// TIA Portal project "Clase4" (V14)
// Equivalente del tutorial 1 del TIA Portal de Youtube

(* hardware
DEVICE "S7-1200 station_1"  S7-1200 Station
   slot 0: "Rack_0"  S7-1200 Rack  Rack  V1.0
   slot 1: "Limon_PLC"  CPU 1214C DC/DC/DC  6ES7 214-1AG40-0XB0  V4.2
DEVICE "S71500/ET200MP station_1"  S7-1500 station
   slot 0: "Rail_0"  Rack  6ES7 590-1***0-0AA0
   slot 1: "Limon 1516"  CPU 1516F-3 PN/DP  6ES7 516-3FN01-0AB0  V2.1
      slot 3: "CPU display_1"  6ES7591-1BA00-0AA0
   slot 2: "DI 32x24VDC HF_1"  DI 32x24VDC HF  6ES7 521-1BL00-0AB0  V2.1
   slot 3: "DQ 32x24VDC/0.5A HF_1"  DQ 32x24VDC/0.5A HF  6ES7 522-1BL01-0AB0  V1.0
   slot 4: "AI 8xU/I/RTD/TC ST_1"  AI 8xU/I/RTD/TC ST  6ES7 531-7KF00-0AB0  V2.1
   slot 5: "AQ 8xU/I HS_1"  AQ 8xU/I HS  6ES7 532-5HF00-0AB0  V2.1
*)

// ===== PLC "Limon_PLC"  CPU 1214C DC/DC/DC =====

VAR_GLOBAL   // PLC tag table "Default tag table"
   "start" AT %I0.0 : Bool;
   "stop" AT %I0.1 : Bool;
   "L1" AT %Q0.0 : Bool;
   "L2" AT %Q0.1 : Bool;
   "variable" AT %M2.0 : Bool;
   "sensor" AT %IW64 : Int;
   "variable_paso" AT %MD4 : Real;
   "lectura" AT %MW8 : Int;
END_VAR

FUNCTION "Arranque_Paro" : Void   // FC1, LAD
TITLE = Arranque y Paro
{ S7_Optimized_Access := 'TRUE' }
VERSION : 0.1
// Demostración de encendido y apagado de una lámpara con enclavamiento.
BEGIN

REGION Network 1: L1
   // Lámpara 1
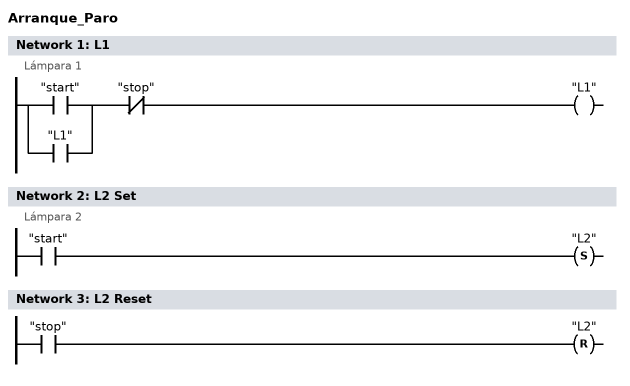
   RUNG wire#powerrail
      Contact( "start" )
      wire#w1
      I_Contact( "stop" )
      Coil( "L1" )
   END_RUNG
   RUNG wire#powerrail
      Contact( "L1" )
   END_RUNG wire#w1
   // the same network as SCL:
   "L1" := ("start" OR "L1") AND NOT "stop";
END_REGION

REGION Network 2: L2 Set
   // Lámpara 2
   RUNG wire#powerrail
      Contact( "start" )
      S_Coil( "L2" )
   END_RUNG
   // the same network as SCL:
   IF "start" THEN "L2" := TRUE; END_IF;
END_REGION

REGION Network 3: L2 Reset
   RUNG wire#powerrail
      Contact( "stop" )
      R_Coil( "L2" )
   END_RUNG
   // the same network as SCL:
   IF "stop" THEN "L2" := FALSE; END_IF;
END_REGION
END_FUNCTION

FUNCTION "Lectura Analogica" : Void   // FC2, LAD
{ S7_Optimized_Access := 'TRUE' }
VERSION : 0.1
BEGIN

REGION Network 1
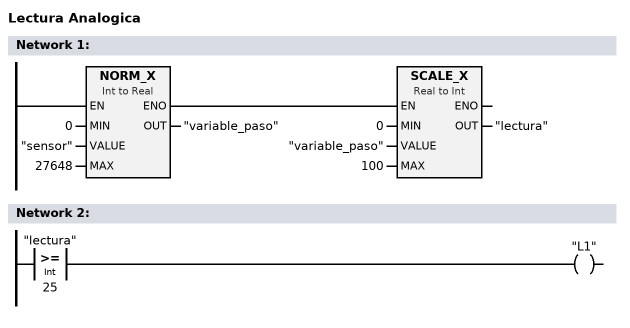
   RUNG wire#powerrail
      { S7_Templates := "[SrcType := Int, DestType := Real]" } Normalize(min := 0, value := "sensor", max := 27648, out => "variable_paso")
      { S7_Templates := "[SrcType := Real, DestType := Int]" } Scale(min := 0, value := "variable_paso", max := 100, out => "lectura")
   END_RUNG
   // the same network as SCL:
   "variable_paso" := NORM_X(MIN := 0, VALUE := "sensor", MAX := 27648);
   "lectura" := SCALE_X(MIN := 0, VALUE := "variable_paso", MAX := 100);
END_REGION

REGION Network 2
   RUNG wire#powerrail
      { S7_Templates := "SrcType := Int" } GE_Contact(in1 := "lectura", in2 := 25)
      Coil( "L1" )
   END_RUNG
   // the same network as SCL:
   "L1" := "lectura" >= 25;
END_REGION
END_FUNCTION

ORGANIZATION_BLOCK "Main"   // OB1, LAD, ProgramCycle
TITLE = "Main Program Sweep (Cycle)"
{ S7_Optimized_Access := 'TRUE' }
VERSION : 0.1
   VAR_INPUT
      Initial_Call : Bool;   // Initial call of this OB
      Remanence : Bool;   // =True, if remanent data are available
   END_VAR
BEGIN

REGION Network 1
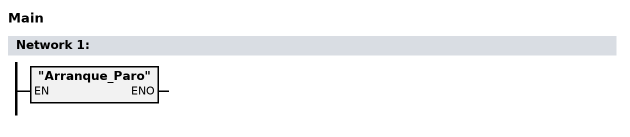
   RUNG wire#powerrail
      "Arranque_Paro"()
   END_RUNG
   // the same network as SCL:
   "Arranque_Paro"();
END_REGION
END_ORGANIZATION_BLOCK

// ===== PLC "Limon 1516"  CPU 1516F-3 PN/DP =====

VAR_GLOBAL   // PLC tag table "Default tag table"
   "inicio" AT %I0.0 : Bool;
   "paro" AT %I0.1 : Bool;
   "L1" AT %Q0.0 : Bool;
   "L2" AT %Q0.1 : Bool;
   "variable" AT %M2.0 : Bool;
   "System_Byte" AT %MB1 : Byte;
   "FirstScan" AT %M1.0 : Bool;
   "DiagStatusUpdate" AT %M1.1 : Bool;
   "AlwaysTRUE" AT %M1.2 : Bool;
   "AlwaysFALSE" AT %M1.3 : Bool;
   "Clock_Byte" AT %MB0 : Byte;
   "Clock_10Hz" AT %M0.0 : Bool;
   "Clock_5Hz" AT %M0.1 : Bool;
   "Clock_2.5Hz" AT %M0.2 : Bool;
   "Clock_2Hz" AT %M0.3 : Bool;
   "Clock_1.25Hz" AT %M0.4 : Bool;
   "Clock_1Hz" AT %M0.5 : Bool;
   "Clock_0.625Hz" AT %M0.6 : Bool;
   "Clock_0.5Hz" AT %M0.7 : Bool;
   "sensor" AT %IW12 : Int;
   "variable de paso" AT %MD18 : Real;
   "lectura" AT %MW22 : Int;
END_VAR

// folder: System blocks/Program resources

DATA_BLOCK "Timer1"   // DB1
{ S7_Optimized_Access := 'TRUE' }
AUTHOR : Simatic
FAMILY : IEC
NAME : IEC_TMR
VERSION : 1.0
// stored: InstanceOfName IEC_TIMER
"IEC_TIMER"
BEGIN
END_DATA_BLOCK

DATA_BLOCK "Timer2"   // DB2
{ S7_Optimized_Access := 'TRUE' }
AUTHOR : Simatic
FAMILY : IEC
NAME : IEC_TMR
VERSION : 1.0
// stored: InstanceOfName IEC_TIMER
"IEC_TIMER"
BEGIN
END_DATA_BLOCK

// folder: (top level)

FUNCTION "Arranque_Paro" : Void   // FC1, LAD
TITLE = Arranque y Paro
{ S7_Optimized_Access := 'TRUE' }
VERSION : 0.1
// Demostración de encendido y apagado de una lámpara con enclavamiento.
BEGIN

REGION Network 1: L1
   // Lámpara 1
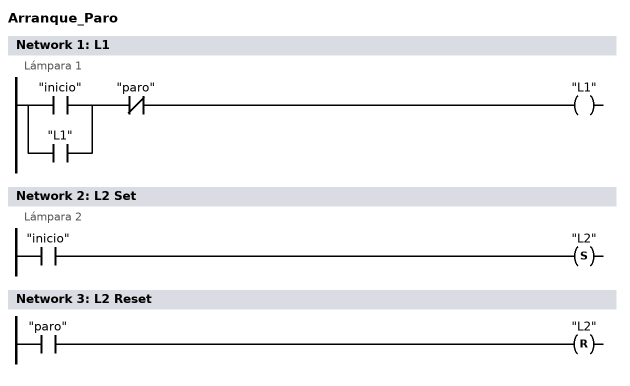
   RUNG wire#powerrail
      Contact( "inicio" )
      wire#w1
      I_Contact( "paro" )
      Coil( "L1" )
   END_RUNG
   RUNG wire#powerrail
      Contact( "L1" )
   END_RUNG wire#w1
   // the same network as SCL:
   "L1" := ("inicio" OR "L1") AND NOT "paro";
END_REGION

REGION Network 2: L2 Set
   // Lámpara 2
   RUNG wire#powerrail
      Contact( "inicio" )
      S_Coil( "L2" )
   END_RUNG
   // the same network as SCL:
   IF "inicio" THEN "L2" := TRUE; END_IF;
END_REGION

REGION Network 3: L2 Reset
   RUNG wire#powerrail
      Contact( "paro" )
      R_Coil( "L2" )
   END_RUNG
   // the same network as SCL:
   IF "paro" THEN "L2" := FALSE; END_IF;
END_REGION
END_FUNCTION

FUNCTION "Blink" : Void   // FC2, LAD
{ S7_Optimized_Access := 'TRUE' }
VERSION : 0.1
   VAR_INPUT
      start : Bool;
      "time" : Time;
   END_VAR
   VAR_OUTPUT
      salida : Bool;
   END_VAR
BEGIN

REGION Network 1
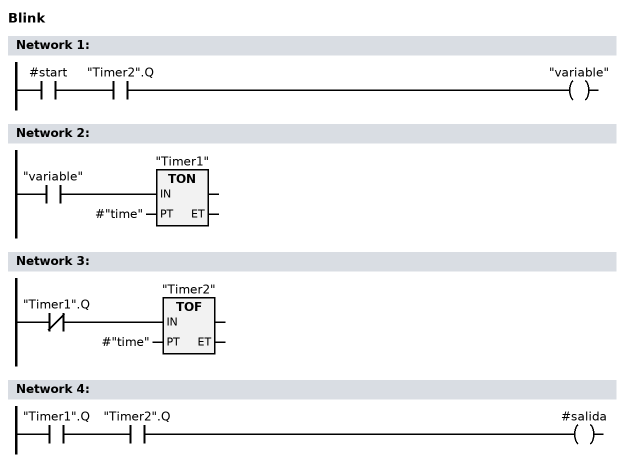
   RUNG wire#powerrail
      Contact( #start )
      Contact( "Timer2".Q )
      Coil( "variable" )
   END_RUNG
   // the same network as SCL:
   "variable" := #start AND "Timer2".Q;
END_REGION

REGION Network 2
   "Timer1".TON(IN := "variable", PT := #"time");
END_REGION

REGION Network 3
   "Timer2".TOF(IN := NOT "Timer1".Q, PT := #"time");
END_REGION

REGION Network 4
   RUNG wire#powerrail
      Contact( "Timer1".Q )
      Contact( "Timer2".Q )
      Coil( #salida )
   END_RUNG
   // the same network as SCL:
   #salida := "Timer1".Q AND "Timer2".Q;
END_REGION
END_FUNCTION

FUNCTION "Lectura Analógica" : Void   // FC3, LAD
{ S7_Optimized_Access := 'TRUE' }
VERSION : 0.1
BEGIN

REGION Network 1
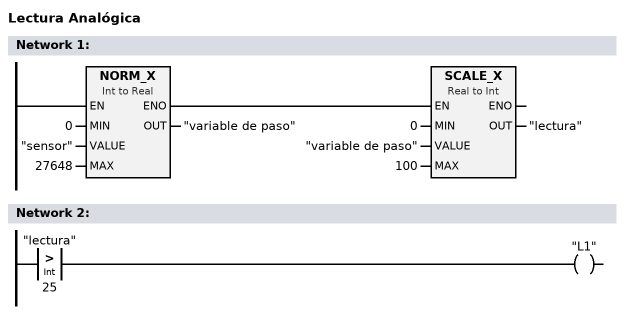
   RUNG wire#powerrail
      { S7_Templates := "[SrcType := Int, DestType := Real]" } Normalize(min := 0, value := "sensor", max := 27648, out => "variable de paso")
      { S7_Templates := "[SrcType := Real, DestType := Int]" } Scale(min := 0, value := "variable de paso", max := 100, out => "lectura")
   END_RUNG
   // the same network as SCL:
   "variable de paso" := NORM_X(MIN := 0, VALUE := "sensor", MAX := 27648);
   "lectura" := SCALE_X(MIN := 0, VALUE := "variable de paso", MAX := 100);
END_REGION

REGION Network 2
   RUNG wire#powerrail
      { S7_Templates := "SrcType := Int" } GT_Contact(in1 := "lectura", in2 := 25)
      Coil( "L1" )
   END_RUNG
   // the same network as SCL:
   "L1" := "lectura" > 25;
END_REGION
END_FUNCTION

ORGANIZATION_BLOCK "Main"   // OB1, LAD, ProgramCycle
TITLE = "Main Program Sweep (Cycle)"
{ S7_Optimized_Access := 'TRUE' }
VERSION : 0.1
   VAR_INPUT
      Initial_Call : Bool;   // Initial call of this OB
      Remanence : Bool;   // =True, if remanent data are available
   END_VAR
BEGIN

REGION Network 1
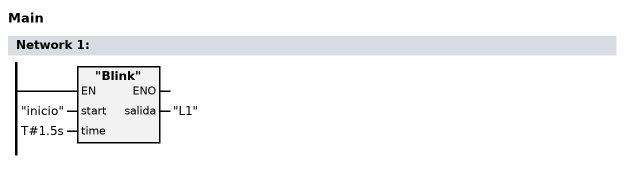
   RUNG wire#powerrail
      "Blink"(start := "inicio", "time" := T#1.5s, salida => "L1")
   END_RUNG
   // the same network as SCL:
   "Blink"(start := "inicio", "time" := T#1.5s, salida => "L1");
END_REGION
END_ORGANIZATION_BLOCK